// TIA Portal V16 export
// export: Created 2022-07-21T09:35:31.6099197Z, ExportSetting WithDefaults, DisplayName Totally Integrated Automation Portal, DisplayVersion V16 Update 4, DisplayName TIA Portal Version Control Interface, DisplayVersion V16 Update 2, DisplayName TIA Portal Openness, DisplayVersion V16 Update 4, DisplayName SINAMICS Startdrive Advanced, DisplayVersion V16 Update 5, DisplayName SINAMICS Startdrive G130, G150, S120, S150, SINAMICS MV, S210, DisplayVersion V16 Update 5, DisplayName SINAMICS Startdrive G110M, G120, G120C, G120D, G120P, G115D, DisplayVersion V16 Update 5, DisplayName STEP 7 Professional, DisplayVersion V16 Update 4, DisplayName STEP 7 Safety, DisplayVersion V16, DisplayName WinCC Advanced, DisplayVersion V16 Update 4
FUNCTION_BLOCK "fbDrive"   // FB36, LAD
TITLE = Drive handling / Obsługa napędu
{ S7_Optimized_Access := 'TRUE' }
VERSION : 0.1
// stored: AutoNumber true, IsIECCheckEnabled false, IsRetainMemResEnabled false, MemoryReserve 100, SetENOAutomatically false, UDAEnableTagReadback false
   VAR_INPUT
      inEnableGeneral : Bool;   // Generalne zezwolenie/urządzenia peryferyjne / General release
      inPowerON : Bool;   // Status zasilania / Power supply status
      InSafetyOK : Bool;   // Safety OK/EStop OK
      inResetEnergySaving : Bool;   // Reset energy saving
      inErrorExt : Bool;   // Zewnętrzny błąd / External alarm
      inRunEnable : Bool;   // Zezwolenie na jazdę / Enable movement
      inEnergySavingTime : Time;   // Czas energy saving / Energy saving time
      inRequestDirectionBackward : Bool;   // Kierunek wstecz / Backward
      inSpeed : Real;   // [m/s]
      inAcceleration { ExternalAccessible := 'False'; ExternalVisible := 'False'; ExternalWritable := 'False'} : Real;   // [m/s²]
      inDeceleration { ExternalAccessible := 'False'; ExternalVisible := 'False'; ExternalWritable := 'False'} : Real;   // [m/s²]
      inPhotocell : "typePhotocell";   // Struktura fotoceli pozycyjnej na przenośniku / Photocell structure
   END_VAR
   VAR_IN_OUT
      ioGroup : "typeGroup";   // Grupa HMI / HMI group
      ioData : "typeConveyor";   // Przenośnik / Conveyor
   END_VAR
   VAR
      sRuntimeEnergySaving : Time;
      sCalculatedRest : Real;
      sTimeSwitchDirectionForward : Time;
      sTimeSwitchDirectionBackward : Time;
   END_VAR
   VAR_TEMP
      tEnable : Bool;
      tRequestEnergySaving : Bool;
      tTimeTillEnergySaving : Time;
      tSpeedPreviousCycle : Real;
      tPowerON : Bool;
      tAutomaticRunConditions : Bool;
   END_VAR
BEGIN

REGION Network 1: Permissions / Sygnały zezwoleń
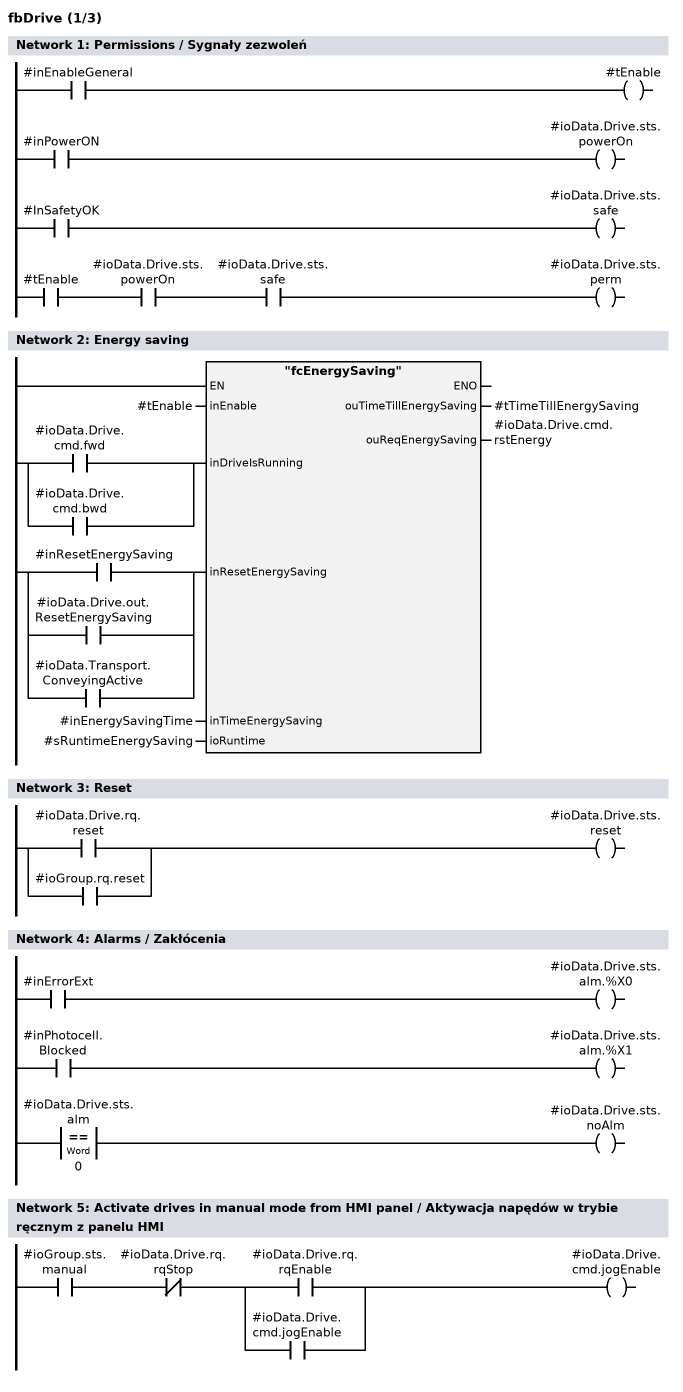
   RUNG wire#powerrail
      Contact( #inEnableGeneral )
      Coil( #tEnable )
   END_RUNG
   RUNG wire#powerrail
      Contact( #inPowerON )
      Coil( #ioData.Drive.sts.powerOn )
   END_RUNG
   RUNG wire#powerrail
      Contact( #InSafetyOK )
      Coil( #ioData.Drive.sts.safe )
   END_RUNG
   RUNG wire#powerrail
      Contact( #tEnable )
      Contact( #ioData.Drive.sts.powerOn )
      Contact( #ioData.Drive.sts.safe )
      Coil( #ioData.Drive.sts.perm )
   END_RUNG
   // the same network as SCL:
   #tEnable := #inEnableGeneral;
   #ioData.Drive.sts.powerOn := #inPowerON;
   #ioData.Drive.sts.safe := #InSafetyOK;
   #ioData.Drive.sts.perm := #tEnable AND #ioData.Drive.sts.powerOn AND #ioData.Drive.sts.safe;
END_REGION

REGION Network 2: Energy saving
   RUNG wire#powerrail
      "fcEnergySaving"(inDriveIsRunning := wire#w1, inResetEnergySaving := wire#w2, inEnable := #tEnable, inTimeEnergySaving := #inEnergySavingTime, ioRuntime := #sRuntimeEnergySaving, ouTimeTillEnergySaving => #tTimeTillEnergySaving, ouReqEnergySaving => #ioData.Drive.cmd.rstEnergy)
   END_RUNG
   RUNG wire#powerrail
      Contact( #ioData.Drive.cmd.fwd )
   END_RUNG wire#w1
   RUNG wire#powerrail
      Contact( #ioData.Drive.cmd.bwd )
   END_RUNG wire#w1
   RUNG wire#powerrail
      Contact( #inResetEnergySaving )
   END_RUNG wire#w2
   RUNG wire#powerrail
      Contact( #ioData.Drive.out.ResetEnergySaving )
   END_RUNG wire#w2
   RUNG wire#powerrail
      Contact( #ioData.Transport.ConveyingActive )
   END_RUNG wire#w2
   // the same network as SCL:
   "fcEnergySaving"(inEnable := #tEnable,
                    inDriveIsRunning := #ioData.Drive.cmd.fwd OR #ioData.Drive.cmd.bwd,
                    inResetEnergySaving := #inResetEnergySaving OR #ioData.Drive.out.ResetEnergySaving OR #ioData.Transport.ConveyingActive,
                    inTimeEnergySaving := #inEnergySavingTime,
                    ioRuntime := #sRuntimeEnergySaving,
                    ouTimeTillEnergySaving => #tTimeTillEnergySaving,
                    ouReqEnergySaving => #ioData.Drive.cmd.rstEnergy);
END_REGION

REGION Network 3: Reset
   RUNG wire#powerrail
      Contact( #ioData.Drive.rq.reset )
      wire#w1
      Coil( #ioData.Drive.sts.reset )
   END_RUNG
   RUNG wire#powerrail
      Contact( #ioGroup.rq.reset )
   END_RUNG wire#w1
   // the same network as SCL:
   #ioData.Drive.sts.reset := #ioData.Drive.rq.reset OR #ioGroup.rq.reset;
END_REGION

REGION Network 4: Alarms / Zakłócenia
   RUNG wire#powerrail
      Contact( #inErrorExt )
      Coil( #ioData.Drive.sts.alm.%X0 )
   END_RUNG
   RUNG wire#powerrail
      Contact( #inPhotocell.Blocked )
      Coil( #ioData.Drive.sts.alm.%X1 )
   END_RUNG
   RUNG wire#powerrail
      { S7_Templates := "SrcType := Word" } EQ_Contact(in1 := #ioData.Drive.sts.alm, in2 := 0)
      Coil( #ioData.Drive.sts.noAlm )
   END_RUNG
   // the same network as SCL:
   #ioData.Drive.sts.alm.%X0 := #inErrorExt;
   #ioData.Drive.sts.alm.%X1 := #inPhotocell.Blocked;
   #ioData.Drive.sts.noAlm := #ioData.Drive.sts.alm = 0;
END_REGION

REGION Network 5: Activate drives in manual mode from HMI panel / Aktywacja napędów w trybie ręcznym z panelu HMI
   RUNG wire#powerrail
      Contact( #ioGroup.sts.manual )
      I_Contact( #ioData.Drive.rq.rqStop )
      wire#w1
      Contact( #ioData.Drive.rq.rqEnable )
      wire#w2
      Coil( #ioData.Drive.cmd.jogEnable )
   END_RUNG
   RUNG wire#w1
      Contact( #ioData.Drive.cmd.jogEnable )
   END_RUNG wire#w2
   // the same network as SCL:
   #ioData.Drive.cmd.jogEnable := #ioGroup.sts.manual AND NOT #ioData.Drive.rq.rqStop AND (#ioData.Drive.rq.rqEnable OR #ioData.Drive.cmd.jogEnable);
END_REGION

REGION Network 6: Move possible in auto/manual / Możliwość jazdy w trybie automatycznym/ tryb ręczny
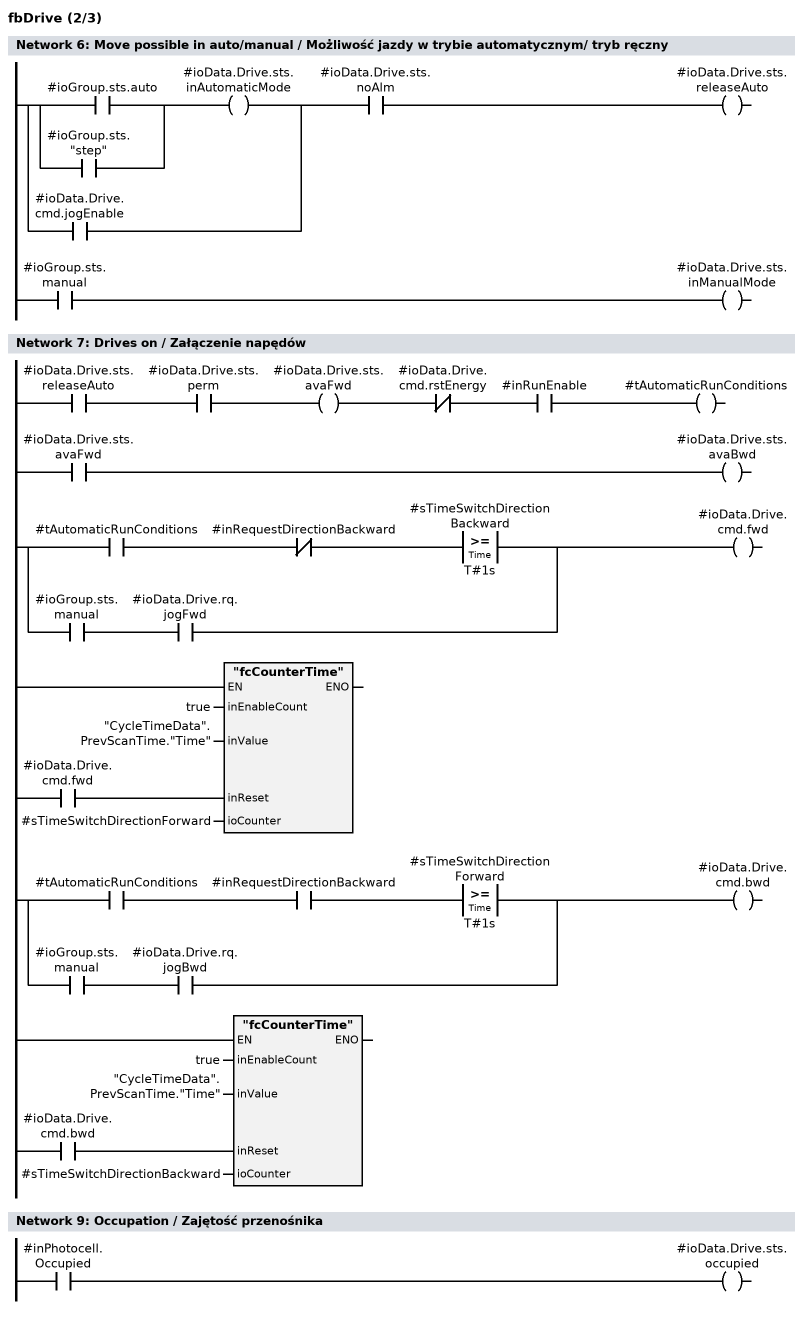
   RUNG wire#powerrail
      Contact( #ioGroup.sts.auto )
      wire#w1
      Coil( #ioData.Drive.sts.inAutomaticMode )
      wire#w2
      Contact( #ioData.Drive.sts.noAlm )
      Coil( #ioData.Drive.sts.releaseAuto )
   END_RUNG
   RUNG wire#powerrail
      Contact( #ioGroup.sts."step" )
   END_RUNG wire#w1
   RUNG wire#powerrail
      Contact( #ioData.Drive.cmd.jogEnable )
   END_RUNG wire#w2
   RUNG wire#powerrail
      Contact( #ioGroup.sts.manual )
      Coil( #ioData.Drive.sts.inManualMode )
   END_RUNG
   // the same network as SCL:
   #ioData.Drive.sts.inAutomaticMode := #ioGroup.sts.auto OR #ioGroup.sts."step";
   #ioData.Drive.sts.releaseAuto := (#ioData.Drive.sts.inAutomaticMode OR #ioData.Drive.cmd.jogEnable) AND #ioData.Drive.sts.noAlm;
   #ioData.Drive.sts.inManualMode := #ioGroup.sts.manual;
END_REGION

REGION Network 7: Drives on / Załączenie napędów
   RUNG wire#powerrail
      Contact( #ioData.Drive.sts.releaseAuto )
      Contact( #ioData.Drive.sts.perm )
      Coil( #ioData.Drive.sts.avaFwd )
      I_Contact( #ioData.Drive.cmd.rstEnergy )
      Contact( #inRunEnable )
      Coil( #tAutomaticRunConditions )
   END_RUNG
   RUNG wire#powerrail
      Contact( #ioData.Drive.sts.avaFwd )
      Coil( #ioData.Drive.sts.avaBwd )
   END_RUNG
   RUNG wire#powerrail
      Contact( #tAutomaticRunConditions )
      I_Contact( #inRequestDirectionBackward )
      { S7_Templates := "SrcType := Time" } GE_Contact(in1 := #sTimeSwitchDirectionBackward, in2 := T#1s)
      wire#w1
      Coil( #ioData.Drive.cmd.fwd )
   END_RUNG
   RUNG wire#powerrail
      Contact( #ioGroup.sts.manual )
      Contact( #ioData.Drive.rq.jogFwd )
   END_RUNG wire#w1
   RUNG wire#powerrail
      "fcCounterTime"(inReset := wire#w2, inEnableCount := true, inValue := "CycleTimeData".PrevScanTime."Time", ioCounter := #sTimeSwitchDirectionForward)
   END_RUNG
   RUNG wire#powerrail
      Contact( #ioData.Drive.cmd.fwd )
   END_RUNG wire#w2
   RUNG wire#powerrail
      Contact( #tAutomaticRunConditions )
      Contact( #inRequestDirectionBackward )
      { S7_Templates := "SrcType := Time" } GE_Contact(in1 := #sTimeSwitchDirectionForward, in2 := T#1s)
      wire#w3
      Coil( #ioData.Drive.cmd.bwd )
   END_RUNG
   RUNG wire#powerrail
      Contact( #ioGroup.sts.manual )
      Contact( #ioData.Drive.rq.jogBwd )
   END_RUNG wire#w3
   RUNG wire#powerrail
      "fcCounterTime"(inReset := wire#w4, inEnableCount := true, inValue := "CycleTimeData".PrevScanTime."Time", ioCounter := #sTimeSwitchDirectionBackward)
   END_RUNG
   RUNG wire#powerrail
      Contact( #ioData.Drive.cmd.bwd )
   END_RUNG wire#w4
   // the same network as SCL:
   #ioData.Drive.sts.avaFwd := #ioData.Drive.sts.releaseAuto AND #ioData.Drive.sts.perm;
   #tAutomaticRunConditions := #ioData.Drive.sts.avaFwd AND NOT #ioData.Drive.cmd.rstEnergy AND #inRunEnable;
   #ioData.Drive.sts.avaBwd := #ioData.Drive.sts.avaFwd;
   #ioData.Drive.cmd.fwd := (#tAutomaticRunConditions AND NOT #inRequestDirectionBackward AND (#sTimeSwitchDirectionBackward >= T#1s)) OR (#ioGroup.sts.manual AND #ioData.Drive.rq.jogFwd);
   "fcCounterTime"(inEnableCount := true,
                   inValue := "CycleTimeData".PrevScanTime."Time",
                   inReset := #ioData.Drive.cmd.fwd,
                   ioCounter := #sTimeSwitchDirectionForward);
   #ioData.Drive.cmd.bwd := (#tAutomaticRunConditions AND #inRequestDirectionBackward AND (#sTimeSwitchDirectionForward >= T#1s)) OR (#ioGroup.sts.manual AND #ioData.Drive.rq.jogBwd);
   "fcCounterTime"(inEnableCount := true,
                   inValue := "CycleTimeData".PrevScanTime."Time",
                   inReset := #ioData.Drive.cmd.bwd,
                   ioCounter := #sTimeSwitchDirectionBackward);
END_REGION

REGION Network 8 (SCL): Calculate speed / Obliczanie prędkości
   REGION Wybór profilu prędkośći
       //-- Sprawdzenie komendy wysterowania napędu
       IF #ioData.Drive.cmd.fwd OR #ioData.Drive.cmd.bwd THEN
           #ioData.Drive.cmd.setpointVelocity := #inSpeed;
       ELSE
           #ioData.Drive.cmd.setpointVelocity := 0.0;
       END_IF;

       //-- Zmiana wartości do obliczeń przy kierunku wstecz
       IF #ioData.Drive.cmd.bwd THEN
           #ioData.Drive.cmd.setpointVelocity *= -1.0;
       END_IF;

   END_REGION;

   REGION Rampa
       //-- Rampa
       #ioData.Drive.cmd.setpointAcceleration := #inAcceleration;
       #ioData.Drive.cmd.setpointDecceleration := #inDeceleration;

   END_REGION ;

   REGION Obliczenia prędkości i dystansu
       //-- Zapamiętanie poprzedniego stanu
       #tSpeedPreviousCycle := #ioData.Drive.sts.actualVelocity;

       //-- Obliczanie prędkośći
       "fcCalculateSpeed"(inAcceleration := #ioData.Drive.cmd.setpointAcceleration,
                          inDeceleration := #ioData.Drive.cmd.setpointDecceleration,
                          inTargetSpeed  := #ioData.Drive.cmd.setpointVelocity,
                          ioCurrentSpeed := #ioData.Drive.sts.actualVelocity);

       //-- Obliczanie dystansu 
       "fcCalculateDistancePerCycle"(inCurrentSpeed     := #ioData.Drive.sts.actualVelocity,
                                     inSpeedPrevScan    := #tSpeedPreviousCycle,
                                     ioRemainder        := #sCalculatedRest,
                                     ouDistancePrevScan => #ioData.Drive.sts.distancePrevScan);
   END_REGION ;

   //-- Napęd jest 'On speed'
   #ioData.Drive.sts.onSpeed := (#ioData.Drive.cmd.fwd OR #ioData.Drive.cmd.bwd)
   AND #ioData.Drive.cmd.setpointVelocity = #ioData.Drive.sts.actualVelocity;
END_REGION

REGION Network 9: Occupation / Zajętość przenośnika
   RUNG wire#powerrail
      Contact( #inPhotocell.Occupied )
      Coil( #ioData.Drive.sts.occupied )
   END_RUNG
   // the same network as SCL:
   #ioData.Drive.sts.occupied := #inPhotocell.Occupied;
END_REGION

REGION Network 10: Interface : ready to receive / Interfejs : gotowość do odbioru
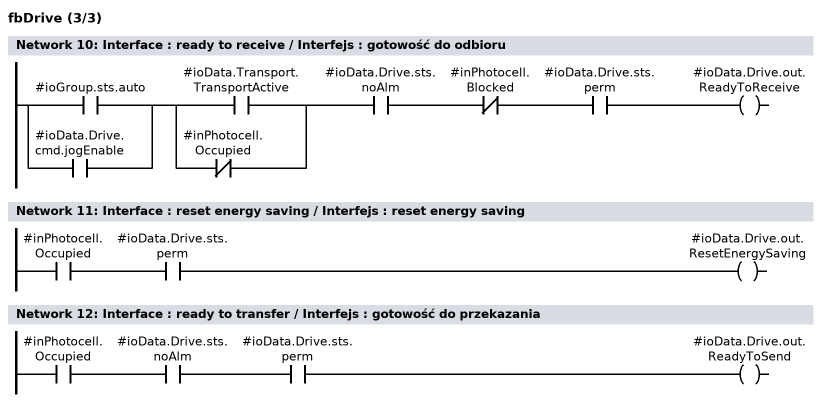
   RUNG wire#powerrail
      Contact( #ioGroup.sts.auto )
      wire#w1
      Contact( #ioData.Transport.TransportActive )
      wire#w2
      Contact( #ioData.Drive.sts.noAlm )
      I_Contact( #inPhotocell.Blocked )
      Contact( #ioData.Drive.sts.perm )
      Coil( #ioData.Drive.out.ReadyToReceive )
   END_RUNG
   RUNG wire#powerrail
      Contact( #ioData.Drive.cmd.jogEnable )
   END_RUNG wire#w1
   RUNG wire#w1
      I_Contact( #inPhotocell.Occupied )
   END_RUNG wire#w2
   // the same network as SCL:
   #ioData.Drive.out.ReadyToReceive := (#ioGroup.sts.auto OR #ioData.Drive.cmd.jogEnable) AND (#ioData.Transport.TransportActive OR NOT #inPhotocell.Occupied) AND #ioData.Drive.sts.noAlm AND NOT #inPhotocell.Blocked AND #ioData.Drive.sts.perm;
END_REGION

REGION Network 11: Interface : reset energy saving / Interfejs : reset energy saving
   RUNG wire#powerrail
      Contact( #inPhotocell.Occupied )
      Contact( #ioData.Drive.sts.perm )
      Coil( #ioData.Drive.out.ResetEnergySaving )
   END_RUNG
   // the same network as SCL:
   #ioData.Drive.out.ResetEnergySaving := #inPhotocell.Occupied AND #ioData.Drive.sts.perm;
END_REGION

REGION Network 12: Interface : ready to transfer / Interfejs : gotowość do przekazania
   RUNG wire#powerrail
      Contact( #inPhotocell.Occupied )
      Contact( #ioData.Drive.sts.noAlm )
      Contact( #ioData.Drive.sts.perm )
      Coil( #ioData.Drive.out.ReadyToSend )
   END_RUNG
   // the same network as SCL:
   #ioData.Drive.out.ReadyToSend := #inPhotocell.Occupied AND #ioData.Drive.sts.noAlm AND #ioData.Drive.sts.perm;
END_REGION
END_FUNCTION_BLOCK
